FUNCTION TryConvert_BYTE_TO_REAL : BOOL
VAR_INPUT
	in : BYTE;
	out : REFERENCE TO REAL;
END_VAR

out := BYTE_TO_REAL(in);
TryConvert_BYTE_TO_REAL := TRUE;

END_FUNCTION

(* stored: Version 1.1.0.1, ProductVersion 3.1.4024.12
   POU TryConvert_BYTE_TO_REAL: Id {548371d1-bfde-4660-9ffc-be036b14e427}, SpecialFunc None *)
